// Mitsubishi GX Developer project: パレット取り外し   PLC: Q02

PROGRAM INISAL
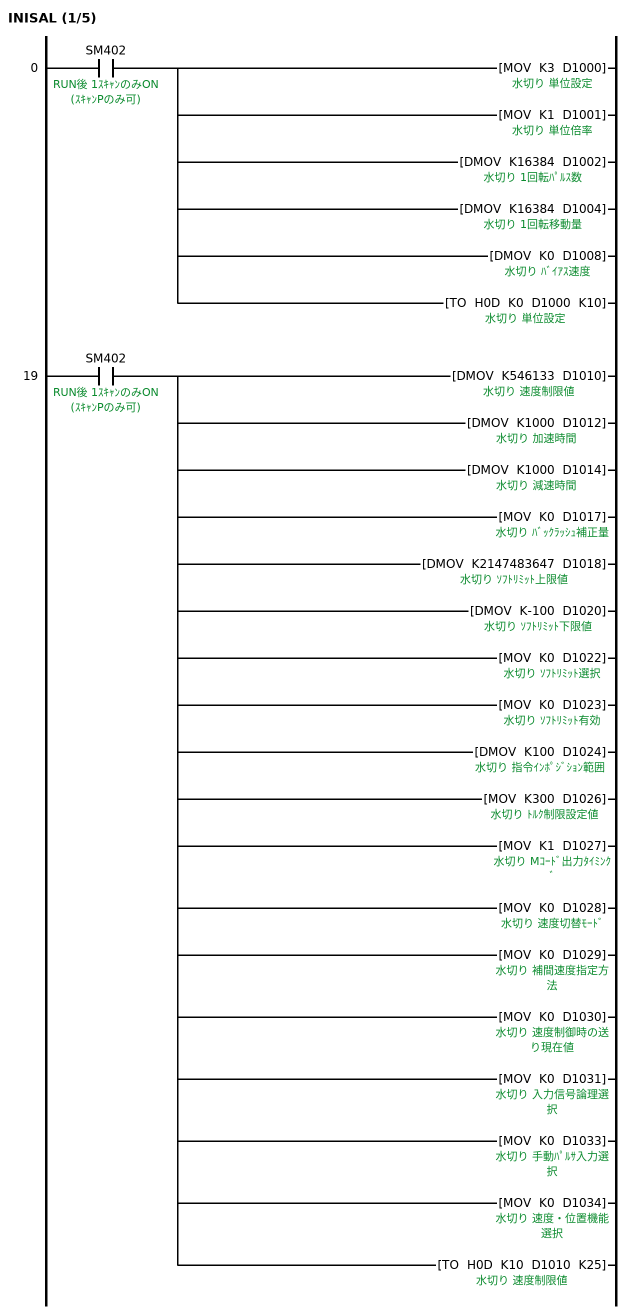
0     LD      SM402  ; RUN後 1ｽｷｬﾝのみON (ｽｷｬﾝPのみ可)
      MOV     K3 D1000  ; 水切り 単位設定
      MOV     K1 D1001  ; 水切り 単位倍率
      DMOV    K16384 D1002  ; 水切り 1回転ﾊﾟﾙｽ数
      DMOV    K16384 D1004  ; 水切り 1回転移動量
      DMOV    K0 D1008  ; 水切り ﾊﾞｲｱｽ速度
      TO      H0D K0 D1000 K10
19    LD      SM402  ; RUN後 1ｽｷｬﾝのみON (ｽｷｬﾝPのみ可)
      DMOV    K546133 D1010  ; 水切り 速度制限値
      DMOV    K1000 D1012  ; 水切り 加速時間
      DMOV    K1000 D1014  ; 水切り 減速時間
      MOV     K0 D1017  ; 水切り ﾊﾞｯｸﾗｯｼｭ補正量
      DMOV    K2147483647 D1018  ; 水切り ｿﾌﾄﾘﾐｯﾄ上限値
      DMOV    K-100 D1020  ; 水切り ｿﾌﾄﾘﾐｯﾄ下限値
      MOV     K0 D1022  ; 水切り ｿﾌﾄﾘﾐｯﾄ選択
      MOV     K0 D1023  ; 水切り ｿﾌﾄﾘﾐｯﾄ有効
      DMOV    K100 D1024  ; 水切り 指令ｲﾝﾎﾟｼﾞｼｮﾝ範囲
      MOV     K300 D1026  ; 水切り ﾄﾙｸ制限設定値
      MOV     K1 D1027  ; 水切り Mｺｰﾄﾞ出力ﾀｲﾐﾝｸﾞ
      MOV     K0 D1028  ; 水切り 速度切替ﾓｰﾄﾞ
      MOV     K0 D1029  ; 水切り 補間速度指定方法
      MOV     K0 D1030  ; 水切り 速度制御時の送り現在値
      MOV     K0 D1031  ; 水切り 入力信号論理選択
      MOV     K0 D1033  ; 水切り 手動ﾊﾟﾙｻ入力選択
      MOV     K0 D1034  ; 水切り 速度・位置機能選択
      TO      H0D K10 D1010 K25
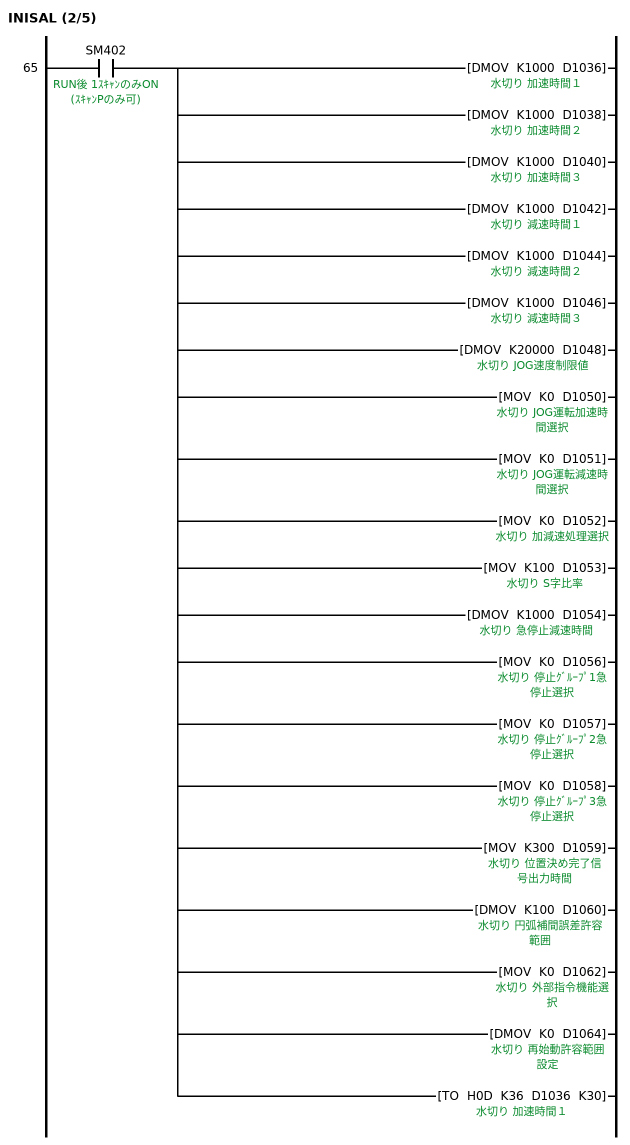
65    LD      SM402  ; RUN後 1ｽｷｬﾝのみON (ｽｷｬﾝPのみ可)
      DMOV    K1000 D1036  ; 水切り 加速時間１
      DMOV    K1000 D1038  ; 水切り 加速時間２
      DMOV    K1000 D1040  ; 水切り 加速時間３
      DMOV    K1000 D1042  ; 水切り 減速時間１
      DMOV    K1000 D1044  ; 水切り 減速時間２
      DMOV    K1000 D1046  ; 水切り 減速時間３
      DMOV    K20000 D1048  ; 水切り JOG速度制限値
      MOV     K0 D1050  ; 水切り JOG運転加速時間選択
      MOV     K0 D1051  ; 水切り JOG運転減速時間選択
      MOV     K0 D1052  ; 水切り 加減速処理選択
      MOV     K100 D1053  ; 水切り S字比率
      DMOV    K1000 D1054  ; 水切り 急停止減速時間
      MOV     K0 D1056  ; 水切り 停止ｸﾞﾙｰﾌﾟ1急停止選択
      MOV     K0 D1057  ; 水切り 停止ｸﾞﾙｰﾌﾟ2急停止選択
      MOV     K0 D1058  ; 水切り 停止ｸﾞﾙｰﾌﾟ3急停止選択
      MOV     K300 D1059  ; 水切り 位置決め完了信号出力時間
      DMOV    K100 D1060  ; 水切り 円弧補間誤差許容範囲
      MOV     K0 D1062  ; 水切り 外部指令機能選択
      DMOV    K0 D1064  ; 水切り 再始動許容範囲設定
      TO      H0D K36 D1036 K30
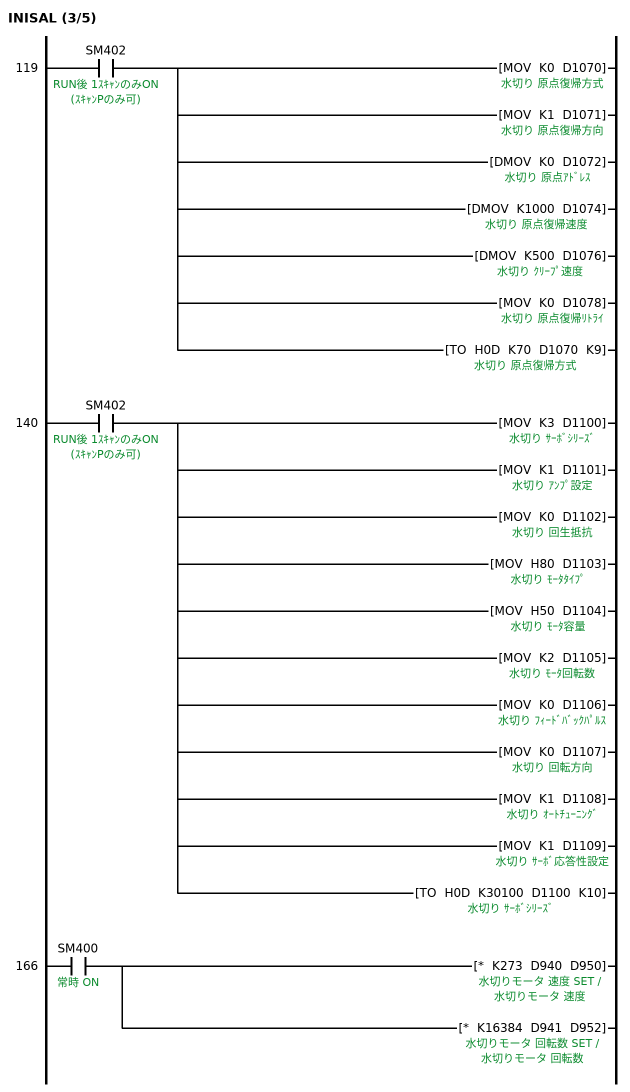
119   LD      SM402  ; RUN後 1ｽｷｬﾝのみON (ｽｷｬﾝPのみ可)
      MOV     K0 D1070  ; 水切り 原点復帰方式
      MOV     K1 D1071  ; 水切り 原点復帰方向
      DMOV    K0 D1072  ; 水切り 原点ｱﾄﾞﾚｽ
      DMOV    K1000 D1074  ; 水切り 原点復帰速度
      DMOV    K500 D1076  ; 水切り ｸﾘｰﾌﾟ速度
      MOV     K0 D1078  ; 水切り 原点復帰ﾘﾄﾗｲ
      TO      H0D K70 D1070 K9
140   LD      SM402  ; RUN後 1ｽｷｬﾝのみON (ｽｷｬﾝPのみ可)
      MOV     K3 D1100  ; 水切り ｻｰﾎﾞｼﾘｰｽﾞ
      MOV     K1 D1101  ; 水切り ｱﾝﾌﾟ設定
      MOV     K0 D1102  ; 水切り 回生抵抗
      MOV     H80 D1103  ; 水切り ﾓｰﾀﾀｲﾌﾟ
      MOV     H50 D1104  ; 水切り ﾓｰﾀ容量
      MOV     K2 D1105  ; 水切り ﾓｰﾀ回転数
      MOV     K0 D1106  ; 水切り ﾌｨｰﾄﾞﾊﾞｯｸﾊﾟﾙｽ
      MOV     K0 D1107  ; 水切り 回転方向
      MOV     K1 D1108  ; 水切り ｵｰﾄﾁｭｰﾆﾝｸﾞ
      MOV     K1 D1109  ; 水切り ｻｰﾎﾞ応答性設定
      TO      H0D K30100 D1100 K10
166   LD      SM400  ; 常時 ON
      *       K273 D940 D950  ; 水切りモータ 速度 SET / 水切りモータ 速度
      *       K16384 D941 D952  ; 水切りモータ 回転数 SET / 水切りモータ 回転数
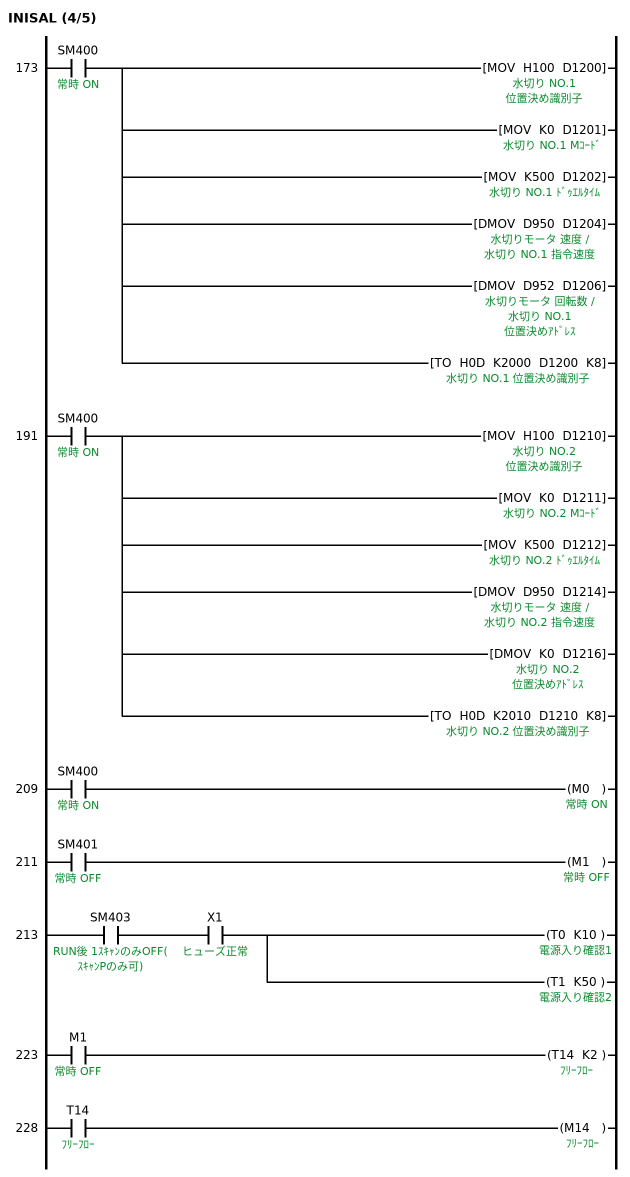
173   LD      SM400  ; 常時 ON
      MOV     H100 D1200  ; 水切り NO.1 位置決め識別子
      MOV     K0 D1201  ; 水切り NO.1 Mｺｰﾄﾞ
      MOV     K500 D1202  ; 水切り NO.1 ﾄﾞｩｴﾙﾀｲﾑ
      DMOV    D950 D1204  ; 水切り NO.1 指令速度
      DMOV    D952 D1206  ; 水切り NO.1 位置決めｱﾄﾞﾚｽ
      TO      H0D K2000 D1200 K8
191   LD      SM400  ; 常時 ON
      MOV     H100 D1210  ; 水切り NO.2 位置決め識別子
      MOV     K0 D1211  ; 水切り NO.2 Mｺｰﾄﾞ
      MOV     K500 D1212  ; 水切り NO.2 ﾄﾞｩｴﾙﾀｲﾑ
      DMOV    D950 D1214  ; 水切り NO.2 指令速度
      DMOV    K0 D1216  ; 水切り NO.2 位置決めｱﾄﾞﾚｽ
      TO      H0D K2010 D1210 K8
209   LD      SM400  ; 常時 ON
      OUT     M0  ; 常時 ON
211   LD      SM401  ; 常時 OFF
      OUT     M1  ; 常時 OFF
213   LD      SM403  ; RUN後 1ｽｷｬﾝのみOFF(ｽｷｬﾝPのみ可)
      AND     X1  ; ヒューズ正常
      OUT     T0 K10  ; 電源入り確認1
      OUT     T1 K50  ; 電源入り確認2
223   LD      M1  ; 常時 OFF
      OUT     T14 K2  ; ﾌﾘｰﾌﾛｰ
228   LD      T14  ; ﾌﾘｰﾌﾛｰ
      OUT     M14  ; ﾌﾘｰﾌﾛｰ
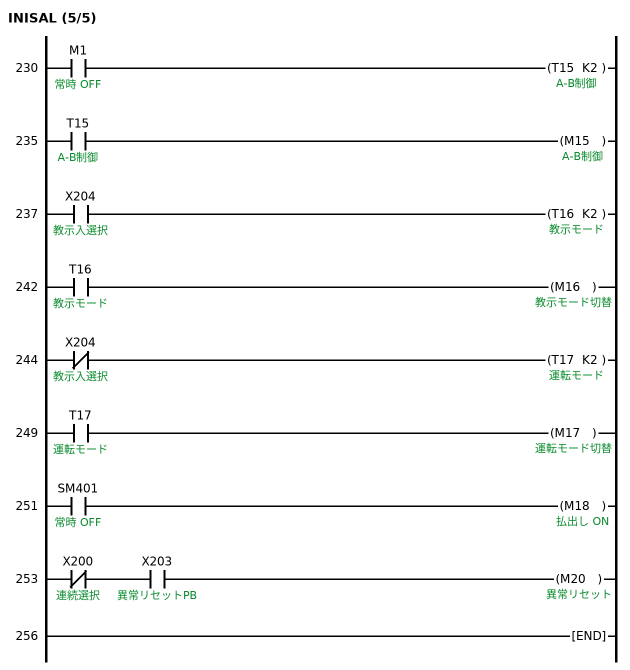
230   LD      M1  ; 常時 OFF
      OUT     T15 K2  ; A-B制御
235   LD      T15  ; A-B制御
      OUT     M15  ; A-B制御
237   LD      X204  ; 教示入選択
      OUT     T16 K2  ; 教示モード
242   LD      T16  ; 教示モード
      OUT     M16  ; 教示モード切替
244   LDI     X204  ; 教示入選択
      OUT     T17 K2  ; 運転モード
249   LD      T17  ; 運転モード
      OUT     M17  ; 運転モード切替
251   LD      SM401  ; 常時 OFF
      OUT     M18  ; 払出し ON
253   LDI     X200  ; 連続選択
      AND     X203  ; 異常リセットPB
      OUT     M20  ; 異常リセット
256   END
END_PROGRAM
